# EPICS substitutions: Db/pciMcorDemo.substitutions
file pciMcorDemoChannel.template
{
	pattern {  chnl }
	{  0 }
	{  1 }
	{  2 }
	{  3 }
	{  4 }
	{  5 }
	{  6 }
	{  7 }
}
